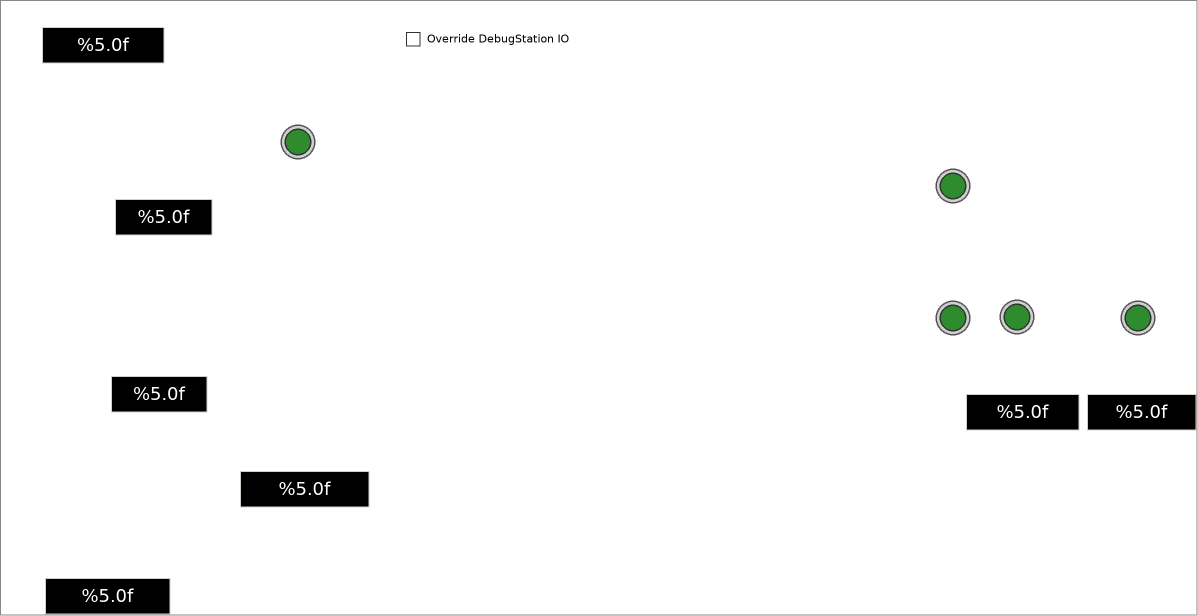
VISUALIZATION HMI_PCW_Monitor  // 1198x616, background image ImageCollection.PCW Flow
    Lamp1 (997,297 40x40), variable: stDebugStation.fbDBStnSeq.stDebugStationDIO.opDBStnLeakFlowPCWValve, style: Lamp-Lamp1-Green
    Textfield (966,394 113x36), "%5.0f", text variable: stDebugStation.fbDBStnSeq.stDebugStationDIO.ipDBStnPCWLeakFlowSensor, input disabled if: TRUE
    Textfield (1087,394 109x36), "%5.0f", text variable: stDebugStation.fbDBStnSeq.stDebugStationDIO.ipDBStnPCWLowFlowSensor, input disabled if: TRUE
    Lamp1 (1118,298 40x40), variable: stDebugStation.fbDBStnSeq.stDebugStationDIO.opDBStnLowFlowPCWValve, style: Lamp-Lamp1-Green
    Lamp1 (933,298 40x40), variable: stDebugStation.fbDBStnSeq.stDebugStationDIO.opDBStnPCWFlowBypassValve, style: Lamp-Lamp1-Green
    Lamp1 (933,166 40x40), variable: stDebugStation.fbDBStnSeq.stDebugStationDIO.opDBStnPCWValve, style: Lamp-Lamp1-Green
    Lamp1 (278,122 40x40), variable: fbDebugColumn.stDebugColumnDIO.opDBColumnPCWValve, style: Lamp-Lamp1-Green
    Textfield (111,376 96x36), "%5.0f", text variable: fbDebugColumn.stDebugColumnDIO.ipDBColumnPCWReturnTemperature, input disabled if: TRUE
    Textfield (45,578 125x36), "%5.0f", text variable: fbDebugColumn.stDebugColumnDIO.ipDBColumnPCWReturnPressure, input disabled if: TRUE
    Textfield (240,471 129x36), "%5.0f", text variable: fbDebugColumn.stDebugColumnDIO.ipDBColumnPCWRegularFlowSensor, input disabled if: TRUE
    Textfield (42,27 122x36), "%5.0f", text variable: fbDebugColumn.stDebugColumnDIO.ipDBColumnPCWSupplyPressure, input disabled if: TRUE
    Textfield (115,199 97x36), "%5.0f", text variable: fbDebugColumn.stDebugColumnDIO.ipDBColumnPCWSupplyTemperature, input disabled if: TRUE
    Rectangle (410,154 428x305)
    Rectangle (468,145 63x323)
    Rectangle (689,144 63x324)
    Rectangle (586,144 63x323)
    Checkbox (404,24 183x30), "Override DebugStation IO"
END_VISUALIZATION

(* stored: Version 1.1.0.1, ProductVersion 3.1.4022.12
   Visu HMI_PCW_Monitor: Id {0b72ae7d-c19d-4eb8-90d7-d7b6afab67c1} *)
